GLOBALCONSTANTS IDs (* Global constants *)
  (* Standard: 61499-1 *)
  (* Version 1.0, 2025-07-24, DEVIASH *)
  VAR_GLOBAL CONSTANT
    ID1 : WSTRING := "topic1";
  END_VAR
END_GLOBALCONSTANTS
